(* IEC 61131-3 sources: CS_4_Aufzugsteuerung/src/Stations/CP112/Steuerung/Class/clsAufzugantrieb, 1 file *)

(* ---- clsAufzugantrieb.st ---- *)
(*!
<Class
	Name               = "clsAufzugantrieb"
	Revision           = "0.0"
	RealtimeTask       = "false"
	CyclicTask         = "true"
	DefCyclictime      = "1 ms"
	BackgroundTask     = "false"
	Sigmatek           = "false"
	OSInterface        = "false"
	HighPriority       = "false"
	Automatic          = "false"
	UpdateMode         = "Prescan"
	SharedCommandTable = "true"
	Objectsize         = "(284,120)">
	<Channels>
		<Server Name="ClassSvr" Visualized="false" Initialize="false" WriteProtected="true" Retentive="false"/>
		<Client Name="cFahrbefehl" Required="false" Internal="false"/>
	</Channels>
</Class>
*)
clsAufzugantrieb : CLASS
  //Servers:
	ClassSvr 	: SvrChCmd_DINT;
  //Clients:
	cFahrbefehl 	: CltChCmd_clsMotorControl;
  //Variables:
		iStep 	: DINT;
  //Functions:

	FUNCTION VIRTUAL GLOBAL CyWork
		VAR_INPUT
			EAX 	: UDINT;
		END_VAR
		VAR_OUTPUT
			state (EAX) 	: UDINT;
		END_VAR;

	FUNCTION GLOBAL FahrtPos
		VAR_INPUT
			xEn 	: DINT;
		END_VAR;

	FUNCTION GLOBAL FahrtNeg
		VAR_INPUT
			xEn 	: DINT;
		END_VAR;
  //Tables:
	FUNCTION @STD
		VAR_OUTPUT
			ret_code	: CONFSTATES;
		END_VAR;
	FUNCTION GLOBAL TAB @CT_;
END_CLASS;

#pragma usingLtd clsMotorControl

FUNCTION VIRTUAL GLOBAL clsAufzugantrieb::CyWork
	VAR_INPUT
		EAX 	: UDINT;
	END_VAR
	VAR_OUTPUT
		state (EAX) 	: UDINT;
	END_VAR

	state := READY;

END_FUNCTION

FUNCTION GLOBAL clsAufzugantrieb::FahrtPos
	VAR_INPUT
		xEn 	: DINT;
	END_VAR

END_FUNCTION

FUNCTION GLOBAL clsAufzugantrieb::FahrtNeg
	VAR_INPUT
		xEn 	: DINT;
	END_VAR

END_FUNCTION
